FUNCTION CheckDivReal : REAL
VAR_INPUT
	divisor		 		: REAL;
END_VAR
VAR
END_VAR

IF divisor = 0 THEN
	CheckRealZeroDiv_ErrCnt := CheckRealZeroDiv_ErrCnt + 1;
	CheckDivReal := 1;
ELSE
	CheckDivReal := divisor;
END_IF

END_FUNCTION

(* stored: Version 1.1.0.1, ProductVersion 3.1.4024.12
   POU CheckDivReal: Id {dac3f469-5340-474e-ad07-623a00451bb7}, SpecialFunc CheckDivReal32 *)
